TYPE ST_System_HOHW_Parameter :
STRUCT
	AutoQuittierung			: BOOL;
END_STRUCT
END_TYPE

(* stored: Version 1.1.0.1, ProductVersion 3.1.4024.9
   DUT ST_System_HOHW_Parameter: Id {690d9a9a-9c25-4d16-8fb7-355357da6df7} *)
